Universal Robots PolyScope program: RC_E7_MOVE_210.urp

Program RC_E7_MOVE_210 (createdIn=3.0.0 lastSavedIn=3.0.0 directory=/programs installation=default)
Robot Program (runOnlyOnce=true motionType=MoveJ speed=1.047198 acceleration=1.396263 useActiveTCP=false)
  'Program generated by RoboDK v4.1.0 for UR3e_HORNO on 05/09/2022 13:22:32'
  'Using nominal kinematics.'
  'Using Ref. UR3_2: p[0.000000, 0.000000, 0.000000, 0.000000, 0.000000, 0.000000]'
  'Using TCP 0208-0001-0001-307-000-3 Horno: p[0.000000, 0.000000, 0.164750, 0.000000, 0.000000, 0.000000]'
  Script: set_tcp(p[0.000000, 0.000000, 0.164750, 0.000000, 0.000000, 0.000000])
  Script: movej([1.452114, -1.409353, -0.955917, -2.344326, 1.570273, 0.520283],0.60000,0.12500,0,0.0000)
